(*
Casts I_Arg as I_BoolArg
*)
FUNCTION ArgToIBoolArg : Result
VAR_INPUT
	iArg		: I_Arg;
END_VAR
VAR_OUTPUT
	iVal		: I_BoolArg;
END_VAR

IF __QUERYINTERFACE(iArg, iVal) THEN
	ArgToIBoolArg := Ok;
END_IF

END_FUNCTION

(* stored: Version 1.1.0.1
   POU ArgToIBoolArg: Id {4a0d7bf2-7557-4fb6-a706-eb119ade3426}, SpecialFunc None *)
